{attribute addProperty BoxType "EK1100-0000-0018"}
{attribute addProperty Id "Beckhoff_EP2xxxEK1122Beckhoff_EP2xxxEK1122_C3355AF127232171798695244"}
{attribute addProperty CRC "2458186430"}
{attribute addProperty SizeInBites "27232"}
{attribute addProperty SizeInBytes "171798695244"}
TYPE Beckhoff_EP2xxx_9284F2BE EXTENDS EK1100_179A0949 :
STRUCT
	{attribute addProperty Name "Beckhoff_EP2xxxEK1122"}
	Beckhoff_EP2xxxEK1122 : Beckhoff_EP2xxxEK1122_C3355AF1;
END_STRUCT
END_TYPE

(* stored: Version 1.2.0.0, ProductVersion 3.1.4024.9
   DUT Beckhoff_EP2xxx_9284F2BE: Id {2b37153b-41e4-465c-b9ee-83d3fab5d630} *)
